//*Hami*
//*Hami* Das Funktion Block liest ein JSON_String von der Ardesse sURi und Schreibt es in OUTPUT value
FUNCTION_BLOCK FB_Get
VAR_INPUT
	bSend				: BOOL;
	sURi : STRING;
	
END_VAR
VAR_IN_OUT
	fbClient			: FB_IotHttpClient;
END_VAR
VAR_OUTPUT
	bBusy				: BOOL;
	bError				: BOOL;
	id					: DINT;
	r_value 			: LREAL;
	value				: DINT;
END_VAR
VAR
	fbHeader: FB_IotHttpHeaderFieldMap ;
	fbRequest			: FB_IotHttpRequest;
	fbJson				: FB_JsonDomParser;
	nState				: UDINT;
	RisingEdge			: R_TRIG;
	
	bGetContentResult	: BOOL;
	sContent			: STRING(511);
	
	bGetJsonResult		: BOOL;
	jsonDoc				: SJsonValue;
	jsonVal				: SJsonValue;
	jsonID				: SJsonValue;
	
	sResultValue		: STRING;
	
	nReqCount			: UDINT;	
	nResCount			: UDINT;
	nValidResCount		: UDINT;
	nErrCount			: UDINT;
	b : BOOL ;
	stReceivedData : ST_ReceivedData ;
	bOnce: BOOL := TRUE ;
	
END_VAR

//*Hami* Authorization einstellen	
	fbHeader.AddField('Authorization', 'Basic RmVsaXg6OGM2OTc2ZTViNTQxMDQxNWJkZTkwOGJkNGRlZTE1ZGZiMTY3YTljODczZmM0YmI4YTgxZjZmMmFiNDQ4YTkxOA==', FALSE);
	fbHeader.AddField('Accept-Language', 'de_DE' , FALSE);
	


//*Hami* hier werden Dateien von sURi als JSON gelesen 
	//RisingEdge(CLK:= bSend );
CASE nState OF
0:	
	//IF RisingEdge.Q THEN 
		IF fbRequest.SendRequest(sURi:=sURi, fbClient:=fbClient, eRequestType:=ETcIotHttpRequestType.HTTP_GET,0, 0, fbHeader) THEN	
	//IF fbRequest.GetJsonDomContent(sURi := sURi , fbClient := fbClient , eRequestType:=ETcIotHttpRequestType.HTTP_GET ,fbJson := fbJson,0) THEN				
			nState:= 1;
			nReqCount:= nReqCount+1;
			bBusy:= TRUE;
			bError:= FALSE;
		END_IF					
	//END_IF
	
//*Hami* hier wird Json_String dekodiert .id und value sind lesbar wenn dateien richtig dekodiert werden
1:
	IF NOT fbRequest.bBusy THEN
		bError:= TRUE;
		IF NOT fbRequest.bError THEN
				bGetContentResult:= fbRequest.GetContent(pContent:= ADR(sContent), nContentSize:= SIZEOF(sContent), bSetNullTermination:= TRUE);
			IF fbRequest.nStatusCode >= 200 AND fbRequest.nStatusCode < 300 THEN
				bGetJsonResult:= FALSE;
				jsonDoc:= fbRequest.GetJsonDomContent(fbJson);
				IF jsonDoc <> 0 THEN
					bGetJsonResult:= TRUE;
					IF fbJson.HasMember(jsonDoc, 'id')  THEN
						jsonID:= fbJson.FindMember(jsonDoc, 'id');
						id := fbJson.GetInt(jsonID);
						IF fbJson.HasMember(jsonDoc, 'value')  THEN
							jsonVal := fbJson.FindMember(jsonDoc, 'value');
							r_value := fbJson.GetDouble(jsonVal);
							value := LREAL_TO_DINT(r_value);
							nValidResCount:= nValidResCount+1;
							bError:= FALSE;						
							IF fbJson.IsString(jsonVal) THEN							
								sResultValue:= fbJson.GetString(jsonVal);									
							END_IF
						END_IF		
					END_IF
				END_IF							
				nResCount:= nResCount+1;			
			END_IF
		END_IF
		nState:= 0;
		bBusy:= FALSE;
		IF bError THEN
			nErrCount:= nErrCount+1;
		END_IF
	END_IF  	
END_CASE

END_FUNCTION_BLOCK

(* stored: Version 1.1.0.1, ProductVersion 3.1.4024.3
   POU FB_Get: Id {ee9d7763-31c2-4203-948c-32ffe0d118d7}, SpecialFunc None *)
